(* IEC 61131-3 sources: ST2CPP/examples/projects/hvac_controller, 5 files *)

(* ---- types.st ---- *)
(* types.st — HVAC 区域控制器类型定义 *)

TYPE
    (* PID 参数结构体 *)
    PID_PARAMS :
    STRUCT
        KP  : REAL;
        KI  : REAL;
        KD  : REAL;
        TS  : REAL;
        MN  : REAL;
        MX  : REAL;
    END_STRUCT;

    (* 区域运行状态 *)
    ZONE_STATE :
    STRUCT
        TEMP      : REAL;
        SETPOINT  : REAL;
        ERROR     : REAL;
        INTEGRAL  : REAL;
        DERIVATIVE : REAL;
        OUTPUT    : REAL;
        MODE      : INT;
        ENABLED   : BOOL;
        ALARM     : BOOL;
        OVRD      : BOOL;
    END_STRUCT;

    (* 传感器量程配置 *)
    SCALE_RANGE :
    STRUCT
        RAW_MIN  : INT;
        RAW_MAX  : INT;
        ENG_MIN  : REAL;
        ENG_MAX  : REAL;
    END_STRUCT;

    (* 区域配置表 *)
    ZONE_CFG :
    STRUCT
        ID          : INT;
        SENSOR_ADDR : INT;
        ACT_ADDR    : INT;
        OCCUPIED    : BOOL;
    END_STRUCT;

    (* 系统告警记录 *)
    ALARM_RECORD :
    STRUCT
        CODE    : INT;
        VALUE   : REAL;
        LATch   : BOOL;
        ACK     : BOOL;
    END_STRUCT;
END_TYPE

(* ---- io_config.st ---- *)
(* io_config.st — HVAC 全局 I/O 映射与配置 *)

VAR_GLOBAL
    (* ─── AI 模拟量输入（12 位 ADC，0-27648 对应 0-10V） ─── *)
    Zone1TempRaw AT %IW0  : INT;
    Zone2TempRaw AT %IW2  : INT;
    Zone3TempRaw AT %IW4  : INT;
    Zone4TempRaw AT %IW6  : INT;
    SupplyTempRaw AT %IW8  : INT;
    ReturnTempRaw AT %IW10 : INT;
    OutsideTempRaw AT %IW12 : INT;
    Zone1HumRaw AT %IW14  : INT;

    (* ─── DI 数字量输入 ─── *)
    StartPB AT %IX0.0   : BOOL;
    StopPB  AT %IX0.1   : BOOL;
    EStop   AT %IX0.2   : BOOL;
    Zone1Occ AT %IX0.3  : BOOL;
    Zone2Occ AT %IX0.4  : BOOL;
    Zone3Occ AT %IX0.5  : BOOL;
    Zone4Occ AT %IX0.6  : BOOL;
    FilterOk AT %IX0.7  : BOOL;

    (* ─── AO 模拟量输出 ─── *)
    Zone1Valve AT %QW0  : INT;
    Zone2Valve AT %QW2  : INT;
    Zone3Valve AT %QW4  : INT;
    Zone4Valve AT %QW6  : INT;
    SupplyValve AT %QW8 : INT;

    (* ─── DO 数字量输出 ─── *)
    SysRun    AT %QX0.0 : BOOL;
    SysAlarm  AT %QX0.1 : BOOL;
    Zone1Heat AT %QX0.2 : BOOL;
    Zone1Cool AT %QX0.3 : BOOL;
    Zone1Fan  AT %QX0.4 : BOOL;
    Zone2Heat AT %QX0.5 : BOOL;
    Zone2Cool AT %QX0.6 : BOOL;
    Zone2Fan  AT %QX0.7 : BOOL;

    (* ─── 全局变量 ─── *)
    SysEnabled    : BOOL := TRUE;
    CycleCount    : DINT := 0;
    GlobalAlarm   : BOOL := FALSE;
    AverageTemp   : REAL := 0.0;
    TotalEnabled  : INT := 0;

    (* ─── 配置常量 ─── *)
    SCALE_10V   : SCALE_RANGE := (RAW_MIN := 0, RAW_MAX := 27648, ENG_MIN := 0.0, ENG_MAX := 100.0);
    SCALE_TEMP  : SCALE_RANGE := (RAW_MIN := 0, RAW_MAX := 27648, ENG_MIN := -40.0, ENG_MAX := 120.0);
    SCALE_HUM   : SCALE_RANGE := (RAW_MIN := 0, RAW_MAX := 27648, ENG_MIN := 0.0, ENG_MAX := 100.0);
END_VAR

(* ---- pid_func.st ---- *)
(* pid_func.st — PID 控制函数 *)

FUNCTION SCALE_AI : REAL
    VAR_INPUT
        RAW     : INT;
        SCALE   : SCALE_RANGE;
    END_VAR
    VAR
        NORM    : REAL;
    END_VAR

    IF RAW > SCALE.RAW_MAX THEN
        NORM := 1.0;
    ELSIF RAW < SCALE.RAW_MIN THEN
        NORM := 0.0;
    ELSE
        NORM := (RAW - SCALE.RAW_MIN) * 1.0 / (SCALE.RAW_MAX - SCALE.RAW_MIN);
    END_IF;

    SCALE_AI := SCALE.ENG_MIN + NORM * (SCALE.ENG_MAX - SCALE.ENG_MIN);
END_FUNCTION

FUNCTION SCALE_AO : INT
    VAR_INPUT
        ENG     : REAL;
        SCALE   : SCALE_RANGE;
    END_VAR
    VAR
        NORM    : REAL;
        RESULT  : INT;
    END_VAR

    NORM := (ENG - SCALE.ENG_MIN) / (SCALE.ENG_MAX - SCALE.ENG_MIN);

    IF NORM > 1.0 THEN
        NORM := 1.0;
    ELSIF NORM < 0.0 THEN
        NORM := 0.0;
    END_IF;

    RESULT := SCALE.RAW_MIN + NORM * (SCALE.RAW_MAX - SCALE.RAW_MIN);
    SCALE_AO := RESULT;
END_FUNCTION

FUNCTION PID_CALC : REAL
    VAR_INPUT
        SP      : REAL;
        PV      : REAL;
        P       : PID_PARAMS;
        DT_VAL  : REAL;
    END_VAR
    VAR
        ERR     : REAL;
        P_TERM  : REAL;
        I_TERM  : REAL;
        D_TERM  : REAL;
        OUTPUT  : REAL;
        INTEGRAL  : REAL := 0.0;
        PREV_ERR : REAL := 0.0;
    END_VAR

    ERR := SP - PV;

    P_TERM := P.KP * ERR;

    INTEGRAL := INTEGRAL + ERR * DT_VAL;
    I_TERM := P.KI * INTEGRAL;

    D_TERM := P.KD * (ERR - PREV_ERR) / DT_VAL;
    PREV_ERR := ERR;

    OUTPUT := P_TERM + I_TERM + D_TERM;

    IF OUTPUT > P.MX THEN
        OUTPUT := P.MX;
    END_IF;
    IF OUTPUT < P.MN THEN
        OUTPUT := P.MN;
    END_IF;

    PID_CALC := OUTPUT;
END_FUNCTION

FUNCTION TEMP_TO_MODE : INT
    VAR_INPUT
        TEMP    : REAL;
        SP      : REAL;
        HYST    : REAL;
    END_VAR

    IF TEMP < SP - HYST THEN
        TEMP_TO_MODE := 1;
    ELSIF TEMP > SP + HYST THEN
        TEMP_TO_MODE := 2;
    ELSE
        TEMP_TO_MODE := 0;
    END_IF;
END_FUNCTION

FUNCTION LIMIT_REAL : REAL
    VAR_INPUT
        X  : REAL;
        MN : REAL;
        MX : REAL;
    END_VAR

    IF X > MX THEN
        LIMIT_REAL := MX;
    ELSIF X < MN THEN
        LIMIT_REAL := MN;
    ELSE
        LIMIT_REAL := X;
    END_IF;
END_FUNCTION

(* ---- zone_fb.st ---- *)
(* zone_fb.st — HVAC 区域控制功能块 *)

FUNCTION_BLOCK ZONE_CTRL
    VAR_INPUT
        RAW_TEMP    : INT;
        OCCUPIED    : BOOL;
        SETPOINT    : REAL;
        ENABLE      : BOOL;
        SCALE       : SCALE_RANGE;
        AO_SCALE    : SCALE_RANGE;
        PID_P       : PID_PARAMS;
    END_VAR
    VAR_OUTPUT
        VALVE_POS   : INT := 0;
        HEAT_OUT    : BOOL := FALSE;
        COOL_OUT    : BOOL := FALSE;
        FAN_OUT     : BOOL := FALSE;
        ZONE_ALARM  : BOOL := FALSE;
        MODE_OUT    : INT := 0;
    END_VAR
    VAR
        STATE       : ZONE_STATE;
        HYSTERESIS  : REAL := 2.0;
        MODE_CMD    : INT := 0;
        MODE_PREV   : INT := 0;
        FAULT_CNT   : INT := 0;
        I           : INT := 0;
    END_VAR

    (* 温度工程值转换 *)
    STATE.TEMP := SCALE_AI(RAW := RAW_TEMP, SCALE := SCALE);

    STATE.SETPOINT := SETPOINT;
    STATE.ENABLED := ENABLE;

    STATE.ERROR := STATE.SETPOINT - STATE.TEMP;

    IF ENABLE THEN
        (* PID 计算 *)
        STATE.OUTPUT := PID_CALC(
            SP := SETPOINT,
            PV := STATE.TEMP,
            P := PID_P,
            DT_VAL := 1.0
        );

        (* 模式选择 *)
        MODE_CMD := TEMP_TO_MODE(TEMP := STATE.TEMP, SP := SETPOINT, HYST := HYSTERESIS);

        (* 状态机 *)
        CASE MODE_CMD OF
            1:
                (* 加热模式 *)
                VALVE_POS := SCALE_AO(ENG := STATE.OUTPUT, SCALE := AO_SCALE);
                HEAT_OUT := STATE.OUTPUT > 0.0;
                COOL_OUT := FALSE;
                FAN_OUT := TRUE;
                MODE_OUT := 1;

            2:
                (* 制冷模式 *)
                VALVE_POS := SCALE_AO(ENG := (0.0 - STATE.OUTPUT), SCALE := AO_SCALE);
                HEAT_OUT := FALSE;
                COOL_OUT := STATE.OUTPUT < -5.0;
                FAN_OUT := TRUE;
                MODE_OUT := 2;

            ELSE
                (* 待机模式 *)
                VALVE_POS := 0;
                HEAT_OUT := FALSE;
                COOL_OUT := FALSE;
                FAN_OUT := MODE_PREV <> 0;
                MODE_OUT := 0;
        END_CASE;

        MODE_PREV := MODE_CMD;

        (* 告警检测 *)
        IF STATE.TEMP > 60.0 OR STATE.TEMP < -10.0 THEN
            FAULT_CNT := FAULT_CNT + 1;
        ELSE
            FAULT_CNT := 0;
        END_IF;

        IF FAULT_CNT >= 3 THEN
            STATE.ALARM := TRUE;
        ELSE
            STATE.ALARM := FALSE;
        END_IF;
    ELSE
        VALVE_POS := 0;
        HEAT_OUT := FALSE;
        COOL_OUT := FALSE;
        FAN_OUT := FALSE;
        MODE_OUT := 0;
        STATE.ALARM := FALSE;
    END_IF;

    ZONE_ALARM := STATE.ALARM;
END_FUNCTION_BLOCK

(* ---- main.st ---- *)
(* main.st — HVAC 主控程序 *)

PROGRAM HVAC_MAIN
    VAR_INPUT
        Start AT %IX1.0  : BOOL;
        Stop  AT %IX1.1  : BOOL;
    END_VAR
    VAR_OUTPUT
        Running AT %QX1.0 : BOOL;
        Fault   AT %QX1.1 : BOOL;
    END_VAR
    VAR
        (* FB 实例 *)
        Z1          : ZONE_CTRL;
        Z2          : ZONE_CTRL;
        Z3          : ZONE_CTRL;
        Z4          : ZONE_CTRL;

        (* 设定值 *)
        HeatSet     : REAL := 22.0;
        CoolSet     : REAL := 24.0;
        EconSet     : REAL := 21.0;

        (* 循环变量 *)
        I           : INT := 0;
        J           : INT := 0;

        (* 运行统计 *)
        ZonesOn     : INT := 0;
        TotalOutput : REAL := 0.0;
        MaxTemp     : REAL := -999.0;
        MinTemp     : REAL := 999.0;
        AnyAlarm    : BOOL := FALSE;

        (* PID 参数 *)
        PID_HOT     : PID_PARAMS := (KP := 2.0, KI := 0.5, KD := 0.1, TS := 1.0, MN := 0.0, MX := 100.0);
        PID_COLD    : PID_PARAMS := (KP := 1.8, KI := 0.3, KD := 0.15, TS := 1.0, MN := -100.0, MX := 0.0);

        (* 状态 *)
        SysMode     : INT := 0;
        OverTemp    : BOOL := FALSE;
        UnderTemp   : BOOL := FALSE;

        (* 测试用 *)
        TestVal     : INT := 0;
        LoopCount   : INT := 0;
        ResultCheck : BOOL := TRUE;
    END_VAR

    (* ─── 系统使能开关 ─── *)
    IF Start AND NOT Stop AND NOT EStop THEN
        SysEnabled := TRUE;
        Running := TRUE;
    ELSE
        SysEnabled := FALSE;
        Running := FALSE;
    END_IF;

    CycleCount := CycleCount + 1;

    (* ─── FOR 循环：处理每个区域 ─── *)
    FOR I := 0 TO 3 BY 1 DO
        IF I = 0 THEN
            (* 区域 1 *)
            Z1(
                RAW_TEMP := Zone1TempRaw,
                OCCUPIED := Zone1Occ,
                SETPOINT := HeatSet,
                ENABLE := SysEnabled,
                SCALE := SCALE_TEMP,
                AO_SCALE := SCALE_10V,
                PID_P := PID_HOT
            );
            Zone1Valve := Z1.VALVE_POS;
            Zone1Heat := Z1.HEAT_OUT;
            Zone1Cool := Z1.COOL_OUT;
            Zone1Fan := Z1.FAN_OUT;

            PRINT("Zone1 active");

            IF Z1.ZONE_ALARM THEN
                GlobalAlarm := TRUE;
            END_IF;

        ELSIF I = 1 THEN
            (* 区域 2 *)
            Z2(
                RAW_TEMP := Zone2TempRaw,
                OCCUPIED := Zone2Occ,
                SETPOINT := CoolSet,
                ENABLE := SysEnabled,
                SCALE := SCALE_TEMP,
                AO_SCALE := SCALE_10V,
                PID_P := PID_COLD
            );
            Zone2Valve := Z2.VALVE_POS;
            Zone2Heat := Z2.HEAT_OUT;
            Zone2Cool := Z2.COOL_OUT;
            Zone2Fan := Z2.FAN_OUT;

        ELSIF I = 2 THEN
            (* 区域 3 *)
            Z3(
                RAW_TEMP := Zone3TempRaw,
                OCCUPIED := Zone3Occ,
                SETPOINT := EconSet,
                ENABLE := SysEnabled,
                SCALE := SCALE_TEMP,
                AO_SCALE := SCALE_10V,
                PID_P := PID_HOT
            );
            Zone3Valve := Z3.VALVE_POS;

        ELSE
            (* 区域 4 *)
            Z4(
                RAW_TEMP := Zone4TempRaw,
                OCCUPIED := Zone4Occ,
                SETPOINT := HeatSet,
                ENABLE := SysEnabled,
                SCALE := SCALE_TEMP,
                AO_SCALE := SCALE_10V,
                PID_P := PID_HOT
            );
            Zone4Valve := Z4.VALVE_POS;
        END_IF;
    END_FOR;

    (* ─── WHILE 循环：统计加热区域数 ─── *)
    J := 0;
    ZonesOn := 0;
    WHILE J <= 3 DO
        IF J = 0 AND Z1.HEAT_OUT THEN
            ZonesOn := ZonesOn + 1;
        ELSIF J = 1 AND Z2.HEAT_OUT THEN
            ZonesOn := ZonesOn + 1;
        ELSIF J = 2 AND Z3.HEAT_OUT THEN
            ZonesOn := ZonesOn + 1;
        ELSIF J = 3 AND Z4.HEAT_OUT THEN
            ZonesOn := ZonesOn + 1;
        END_IF;
        J := J + 1;
    END_WHILE;

    (* ─── REPEAT 循环：计算平均温度 ─── *)
    TotalOutput := 0.0;
    I := 0;
    REPEAT
        TotalOutput := TotalOutput + 25.0;
        I := I + 1;
    UNTIL I >= 4
    END_REPEAT;

    AverageTemp := TotalOutput / 4.0;

    (* ─── CASE 系统模式选择 ─── *)
    SysMode := 0;
    IF Z1.HEAT_OUT OR Z2.HEAT_OUT THEN
        SysMode := 1;
    END_IF;
    IF Z1.COOL_OUT OR Z2.COOL_OUT THEN
        SysMode := 2;
    END_IF;

    CASE SysMode OF
        1:
            SysRun := TRUE;
        2:
            SysRun := TRUE;
        ELSE
            SysRun := ZonesOn > 0;
    END_CASE;

    (* ─── 告警汇总逻辑 ─── *)
    AnyAlarm := Z1.ZONE_ALARM OR Z2.ZONE_ALARM OR Z3.ZONE_ALARM OR Z4.ZONE_ALARM;
    SysAlarm := AnyAlarm;
    Fault := AnyAlarm;

    (* ─── EXIT/CONTINUE 测试 ─── *)
    TestVal := 0;
    FOR I := 0 TO 10 BY 1 DO
        IF I = 5 THEN
            CONTINUE;
        END_IF;
        TestVal := TestVal + 1;
        IF I > 8 THEN
            EXIT;
        END_IF;
    END_FOR;

    (* ─── 复杂表达式测试 ─── *)
    OverTemp := (Z1.STATE.TEMP > 50.0 AND Z1.STATE.TEMP <> -999.0) OR Z1.ZONE_ALARM;
    UnderTemp := Z1.STATE.TEMP < -5.0 AND NOT Z1.ZONE_ALARM;

    TotalEnabled := 0;
    IF Zone1Occ THEN TotalEnabled := TotalEnabled + 1; END_IF;
    IF Zone2Occ THEN TotalEnabled := TotalEnabled + 1; END_IF;
    IF Zone3Occ THEN TotalEnabled := TotalEnabled + 1; END_IF;
    IF Zone4Occ THEN TotalEnabled := TotalEnabled + 1; END_IF;

    LoopCount := I * 10 + J;
    ResultCheck := LoopCount > 0 AND TestVal = 9;

    (* ─── 集成断言验证 ─── *)
    PRINT("HVAC cycle complete");
    ASSERT(LoopCount >= 0);
    ASSERT(SysEnabled OR NOT Running);
    ASSERT(ResultCheck OR AnyAlarm);
END_PROGRAM
